// SIMATIC S7-200 project (STEP 7-Micro/WIN), CPU 224XP REL 02.01

SYMBOL_TABLE USUARIO1
PARO_1           I0.0
PAR0_2           I0.1
MARCHA_1         I0.2
MARCHA_2         I0.3
MARCHA_3         I0.4
E1               Q0.0
E2               Q0.1
E3               Q0.2
E4               Q0.3
E5               Q0.4
END_SYMBOL_TABLE

ORGANIZATION_BLOCK PRINCIPAL:OB1
TITLE=COMENTARIOS DEL PROGRAMA
BEGIN
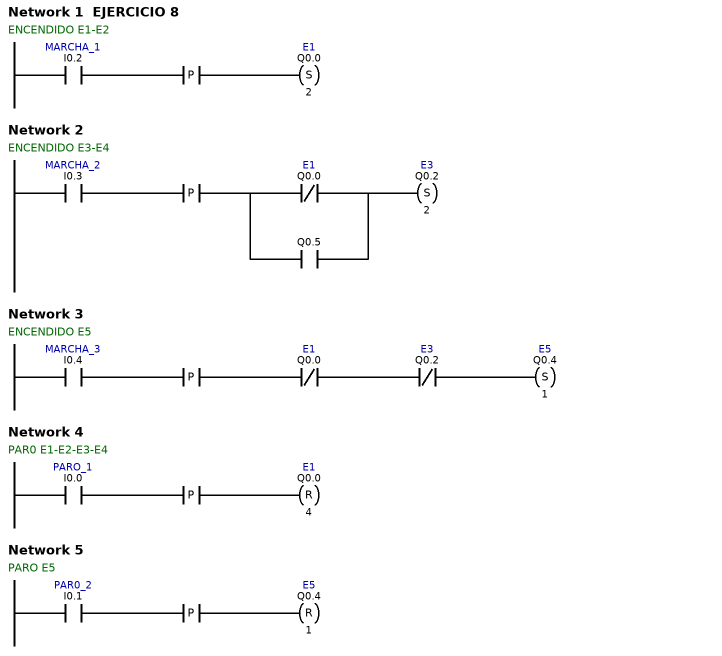
Network 1 // EJERCICIO 8
// ENCENDIDO E1-E2
LD     MARCHA_1:I0.2
EU
S      E1:Q0.0, 2
Network 2
// ENCENDIDO E3-E4
LD     MARCHA_2:I0.3
EU
LDN    E1:Q0.0
O      Q0.5
ALD
S      E3:Q0.2, 2
Network 3
// ENCENDIDO E5
LD     MARCHA_3:I0.4
EU
AN     E1:Q0.0
AN     E3:Q0.2
S      E5:Q0.4, 1
Network 4
// PAR0 E1-E2-E3-E4
LD     PARO_1:I0.0
EU
R      E1:Q0.0, 4
Network 5
// PARO E5
LD     PAR0_2:I0.1
EU
R      E5:Q0.4, 1
END_ORGANIZATION_BLOCK
